{attribute addProperty BoxType "EL5151-0000-0016"}
{attribute addProperty Id "Enable_latch_CAT %Q*BOOL811Enable_latch_extern_on_positive_edgeAT %Q*BOOL812Set_counterAT %Q*BOOL813Enable_latch_extern_on_negative_edgeAT %Q*BOOL814Set_counter_valueAT %Q*UDINT32417"}
{attribute addProperty CRC "2419543123"}
{attribute addProperty SizeInBites "64"}
{attribute addProperty SizeInBytes "8"}
TYPE ENC_Outputs_90374C53 :
STRUCT
	{attribute addProperty Name "Enable_latch_C"}
	Enable_latch_C AT %Q* : BOOL;
	{attribute addProperty Name "Enable_latch_extern_on_positive_edge"}
	Enable_latch_extern_on_positive_edge AT %Q* : BOOL;
	{attribute addProperty Name "Set_counter"}
	Set_counter AT %Q* : BOOL;
	{attribute addProperty Name "Enable_latch_extern_on_negative_edge"}
	Enable_latch_extern_on_negative_edge AT %Q* : BOOL;
	{attribute addProperty Name "Set_counter_value"}
	Set_counter_value AT %Q* : UDINT;
END_STRUCT
END_TYPE

(* stored: Version 1.2.0.0, ProductVersion 3.1.4024.9
   DUT ENC_Outputs_90374C53: Id {3f859fb4-7d88-4159-b4a5-2bb45e3789e2} *)
